FUNCTION_BLOCK FB_AmbientAir 
VAR_INPUT
END_VAR
VAR_OUTPUT
END_VAR
VAR
	ftemp_sin: OSCAT.GEN_SIN:= ( PT := T#10S,
								     AM := 7,
								     OS := 12,
								     DL:= 0); 
END_VAR

METHOD Run 
VAR_INPUT
END_VAR
ftemp_sin();
GVL.fTempAmbAir := ftemp_sin.Out;
END_METHOD

END_FUNCTION_BLOCK

(* stored: Version 1.1.0.1, ProductVersion 3.1.4024.3
   POU FB_AmbientAir: Id {90d51716-db66-4a5f-aa64-9deae95092df}, SpecialFunc None
   Method Run: Id {cbf9f38b-8652-4b83-8fba-69d0b7cd88b3} *)
